# EPICS StreamDevice protocol: sampleApp/protocol/VICI.proto
# VICI Valco Protocol
# A. Wallace 2014-3-18

Terminator = CR;
ReplyTimeout  =  800;
ReadTimeout   =  100;
WriteTimeout  =  100;
ExtraInput    =  Ignore;

## Generic get/set
# \$1=command, \$2=conversion

ParamGet{ out "0\$1"; in "0\$1%2d"; }
SParamGet{ out "0\$1"; in "0\$1%s"; }
VerGet{ out "\$1"; in "%s"; }
ParamSet{ out "\$1%i"; }

NMoveCW		{ out "0CW%i";	}
NMoveCCW	{ out "0CC%i";	}

2PosSet	{ out "GO%{A|B}";	}
2PosGet	{ out "CP"; in "CP%{A|B}";	}
#For commands that do not pass any information
BlankOut{ out "\$1"; }

#GET_BY       { out "1PR BY";        in "%s";        wait 25; }
